FUNCTION_BLOCK PUBLIC FB_LampUpDown EXTENDS FB_Lamp
VAR
	nLightLevel			: BYTE(0..100);
END_VAR

// Reduces the control value by 5 in the range of 10 to 100.
METHOD PUBLIC DimDown
IF (nLightLevel >= 15) THEN
	OneStepDown();
	OneStepDown();
	OneStepDown();
	OneStepDown();
	OneStepDown();
END_IF
END_METHOD

// Increments the control value by 5 in the range of 10 to 100.
METHOD PUBLIC DimUp
IF (nLightLevel <= 95) THEN	
	OneStepUp();
	OneStepUp();
	OneStepUp();
	OneStepUp();
	OneStepUp();
END_IF
END_METHOD

// Sets the control value to 0.
METHOD PUBLIC Off
IF (nLightLevel > 0) THEN
	OnOff();
END_IF
END_METHOD

// Sets the control value to 100.
METHOD PUBLIC On
IF (nLightLevel = 0) THEN
	OnOff();
END_IF
END_METHOD

// Reduces the control value by 1 in the range of 10 to 100.
METHOD PUBLIC OneStepDown
nLightLevel := nLightLevel - 1;
IF (nLightLevel < 10) THEN
	nLightLevel := 10;
END_IF
IF (_ipObserver <> 0) THEN
	_ipObserver.Update(nLightLevel);
END_IF
END_METHOD

// Increments the control value by 1 in the range of 10 to 100.
METHOD PUBLIC OneStepUp
nLightLevel := nLightLevel + 1;
IF (nLightLevel > 100) THEN
	nLightLevel := 100;
END_IF
IF (_ipObserver <> 0) THEN
	_ipObserver.Update(nLightLevel);
END_IF
END_METHOD

// Toggles the control value between 0 and 100.
METHOD PUBLIC OnOff
IF (nLightLevel > 0) THEN
	nLightLevel := 0;
ELSE
	nLightLevel := 100;
END_IF
IF (_ipObserver <> 0) THEN
	_ipObserver.Update(nLightLevel);
end_IF
END_METHOD

END_FUNCTION_BLOCK

(* stored: Version 1.1.0.1, ProductVersion 3.1.4024.9
   POU FB_LampUpDown: Id {e5938590-1890-43a0-ba86-32547ab377e2}, SpecialFunc None
   Method DimDown: Id {f433ba23-f42e-4cab-9ef3-5e4194ea6188}
   Method DimUp: Id {ade1dbbc-7478-4536-897c-2d3c2ded4722}
   Method Off: Id {868806eb-f2e3-4d33-9bab-570b2abb5487}
   Method On: Id {8e9c39de-7158-4dff-b672-3b0f3333d1ca}
   Method OneStepDown: Id {eccc8046-24a1-4940-82a7-bde5c3e6c0ab}
   Method OneStepUp: Id {bdc89d87-e6d0-409f-9392-70820315cfad}
   Method OnOff: Id {4e5634f0-9545-430f-86b8-452bc4855175} *)
